PROGRAM PRG_PID_CALL
VAR
END_VAR

END_PROGRAM

(* stored: Version 1.1.0.1, ProductVersion 3.1.4024.13
   POU PRG_PID_CALL: Id {e7fc84ae-b95c-477c-b1bf-9630c0dddc70}, SpecialFunc None *)
